FUNCTION_BLOCK XtsDisableSequence EXTENDS TaskBase
VAR_INPUT
END_VAR
VAR_OUTPUT
END_VAR
VAR
	_collisionGroup : ICollisionGroup;
	removeAllAxes : RemoveAllMoverFromGroup(_collisionGroup);
	grpStop : StopMoverGroup(_collisionGroup);
	DisableTrigger: BOOL;
	moverNumbers : UINT := 1;
	AllMoversDisabled: BOOL;	
	Logger : TcMessage_Ext;
	arrMovers : ARRAY[1..SystemParameters.NumberOfMovers] OF IMover;
END_VAR

{analysis -2}

METHOD Abort : BOOL
VAR
	RemoveAxisAbortResult : BOOL;
	GroupAbortResult : BOOL;
END_VAR
DisableTrigger := FALSE;
State := 0;
RemoveAxisAbortResult := removeAllAxes.Abort();
GroupAbortResult := grpStop.Abort();
Abort := RemoveAxisAbortResult AND GroupAbortResult;
END_METHOD

METHOD Cycle : HRESULT
VAR_INPUT
END_VAR
Cycle := S_OK;
CASE State OF
	0:
		IF DisableTrigger THEN
			Cycle := S_PENDING;
			DisableTrigger := FALSE;
			_Busy := TRUE;
			_Done := FALSE;
			_Error := FALSE;
			IF _collisionGroup.GroupState = CAGroupStatus.mcGroupStateMoving THEN
				Logger.Send(TC_EVENTS.XtsCaGroupEvents.CAGroupStop,'');
				grpStop.Execute();
				State := 10;
			ELSE
				State := 20;
				removeAllAxes.RemoveAllMover();
				Logger.Send(TC_EVENTS.XtsCaGroupEvents.CaGroupRemoveMovers,'');
			END_IF
		END_IF
		
	10:
		IF grpStop.Done THEN
			State := 20;
			Logger.Send(TC_EVENTS.XtsCaGroupEvents.CaGroupRemoveMovers,'');
			removeAllAxes.RemoveAllMover();
		END_IF
	
	20:
		IF removeAllAxes.Done THEN
			FOR moverNumbers := 1 TO SystemParameters.NumberOfMovers DO
				arrMovers[moverNumbers].IdentInGroup := 0;
				arrMovers[moverNumbers].DisableAxis();
			END_FOR
			State := 30;
		END_IF
		
	30:
		AllMoversDisabled := TRUE;
		FOR moverNumbers := 1 TO SystemParameters.NumberOfMovers DO
			AllMoversDisabled := TRUE AND NOT arrMovers[moverNumbers].isEnabled();
		END_FOR
		IF AllMoversDisabled THEN
			Logger.Send(TC_EVENTS.XtsCaGroupEvents.AllMoversDisabled,'');
			State := 40;
			_collisionGroup.Disable();
			Logger.Send(TC_EVENTS.XtsCaGroupEvents.CAGroupDisable,'');
		END_IF
	40:
		IF _collisionGroup.GroupState = CAGroupStatus.mcGroupStateErrorStop THEN
			_collisionGroup.Reset();
			Logger.Send(TC_EVENTS.XtsCaGroupEvents.CAGroupReset,'');
		END_IF	
		State := 50;
		
	50:
		IF _collisionGroup.GroupState = 1 THEN
			State := 0;
			grpStop.Deceleration := Tc3_Mc3Definitions.MC_DEFAULT;
			grpStop.Jerk := Tc3_Mc3Definitions.MC_DEFAULT;
			Cycle := S_OK;
			_Busy := FALSE;
			_Done := TRUE;
		END_IF
	ELSE
		Cycle := E_FAIL;
END_CASE

removeAllAxes.Cycle();
grpStop.Cycle();
END_METHOD

METHOD Disable : BOOL
VAR_INPUT
END_VAR
DisableTrigger := true;
END_METHOD

METHOD FB_init : BOOL
VAR_INPUT
	bInitRetains : BOOL; // if TRUE, the retain variables are initialized (warm start / cold start)
	bInCopyCode : BOOL;  // if TRUE, the instance afterwards gets moved into the copy code (online change)
	MyCaGroup : ICollisionGroup;
END_VAR
_collisionGroup := MyCaGroup;
removeAllAxes.FB_init(FALSE, FALSE, MyCaGroup := MyCaGroup);
grpStop.FB_init(FALSE,FALSE,CAGroup := MyCaGroup);
END_METHOD

PROPERTY MoverArray : array[1..SystemParameters.NumberOfMovers] of IMover
GET
MoverArray := arrMovers;
END_GET
SET
arrMovers := MoverArray;
END_SET
END_PROPERTY

METHOD SetEmergencyDynamics : BOOL
VAR_INPUT
END_VAR
grpStop.Deceleration := Tc3_Mc3Definitions.MC_MAXIMUM;
grpStop.Jerk := Tc3_Mc3Definitions.MC_MAXIMUM;
END_METHOD

END_FUNCTION_BLOCK

(* stored: Version 1.1.0.1, ProductVersion 3.1.4024.12
   POU XtsDisableSequence: Id {da9628bf-0fcc-432f-b10d-3ad4dd4b7f24}, SpecialFunc None
   Method Abort: Id {86211cf7-3baa-4942-994c-481ee3b2466c}
   Method Cycle: Id {981b7190-eb15-4a0a-8875-0afb334ed36e}
   Method Disable: Id {024bbd18-8e3c-4aa1-9d04-45454423df20}
   Method FB_init: Id {5c39a8d0-8d47-4b10-ae0c-53e63f445cbe}
   Property MoverArray: Id {5eeee228-c90c-4059-b15e-d4f3141abdbb}
   Get Get: Id {b10eaf89-7079-42df-9644-c9a26f75907c}
   Set Set: Id {c98462cb-d524-483d-aa6e-1ec06568f609}
   Method SetEmergencyDynamics: Id {e46d706c-c452-462f-8599-1eb3f1547e4f} *)
